{attribute 'no_check'}
// description of Slave Job (data structure)
FUNCTION_BLOCK ModbusJob	
VAR_INPUT
	FunctionCode		:	BYTE;
	StartAddress		:	WORD;
	Quantity			:	WORD;
	Valid				:	BOOL;
	Timestamp			:	DATE_AND_TIME;
END_VAR
VAR_OUTPUT
END_VAR
VAR
END_VAR

;

METHOD PUBLIC init : BOOL //Return value = TRUE if execution finished
VAR_INPUT
END_VAR
	functionCode											:= 0;
	startAddress											:= 0;
	valid													:= FALSE;
	MEMSET(ADR(quantity), 16#0, SIZEOF(quantity));	
	MEMSET(ADR(timeStamp), 16#0, SIZEOF(timeStamp));
	Init													:= TRUE;
END_METHOD

END_FUNCTION_BLOCK

(* stored: Version 1.1.0.1, ProductVersion 3.1.4024.3
   POU ModbusJob: Id {e1f85871-53c6-43b4-bcca-cc8cba56ee95}, SpecialFunc None
   Method init: Id {8b5e6970-f463-47cc-ac38-e062be9549a4} *)
